FUNCTION_BLOCK ABSTRACT FB_Parent
VAR
	sOutput : STRING;
END_VAR

METHOD ABSTRACT Eat
VAR_INPUT
END_VAR
END_METHOD

METHOD FB_init : BOOL
VAR_INPUT
	bInitRetains : BOOL; // if TRUE, the retain variables are initialized (warm start / cold start)
	bInCopyCode : BOOL;  // if TRUE, the instance afterwards gets moved into the copy code (online change)
END_VAR
sOutput := 'I am in the parent class';
END_METHOD

METHOD ABSTRACT Greet  
VAR_INPUT
END_VAR
END_METHOD

METHOD Greeting
VAR_INPUT
END_VAR
sOutput := 'Greetings of the day : ';
END_METHOD

END_FUNCTION_BLOCK

(* stored: Version 1.1.0.1, ProductVersion 3.1.4024.16
   POU FB_Parent: Id {dea553f7-b534-44d6-ad91-d48fab43a13d}, SpecialFunc None
   Method Eat: Id {76cac19c-1079-4b8e-a563-a1eeaac78e54}
   Method FB_init: Id {146764ac-048e-4fbc-950b-fbcf7acad751}
   Method Greet: Id {cdde60cd-3ce3-48a0-a000-7926ce0b471b}
   Method Greeting: Id {63d452c3-ae38-4372-9d94-47bda443a9ad} *)
